{attribute 'no_assign'}
{attribute 'qualified_only'}
VAR_GLOBAL
    TcUnitRunner : FB_TcUnitRunner;

    (* Indication of whether the last instantiated test suite has an assert instance created *)
    TestSuiteIsRegistered : BOOL;

    (* Pointer to current test suite being called *)
    CurrentTestSuiteBeingCalled : POINTER TO FB_TestSuite;

    (* Current name of test being called *)
    CurrentTestNameBeingCalled : Tc2_System.T_MaxString;

    (* This is a flag that indicates that the current test should be ignored, and
       thus that all assertions under it should be ignored as well. A test can be ignored either
       because the user has requested so, or because the test is a duplicate name *)
    IgnoreCurrentTest : BOOL;

    (* The assert function block instance should be 1:1 mapped to
       the test suite instance path. *)
    AmountOfInitializedTestSuites : UINT := 0;
    TestSuiteAddresses : ARRAY[1..GVL_Constants.MaxAmountOfTestSuites] OF POINTER TO FB_TestSuite;
END_VAR

(* stored: Version 1.1.0.1, ProductVersion 3.1.4022.9
   GVL GVL: Id {78472b76-c9a4-4b27-a580-8e7898edc3d7} *)
